{attribute 'qualified_only'}
VAR_GLOBAL
	// Schnittstellenvariablen 
		// System: 
		SystemState								:eSystemState; 
		SystemCommand							:eSystemCommand; 
		Error									:BOOL;
		
		// Kontrollvariablen: 
		Reset									:BOOL;
		
		// Prozessvariablen
		eKraftLimitValue						:sKraftVariablen;
		eKraftErreichtValue						:sKraftVariablen;
		
		
		// SkillStates
		
		// ObjectStates
		Robot_State								:eObjectState;
		Greifer_State							:eObjectState;
		Sensor_State							:eObjectState;
		
			
		
		
		
END_VAR

(* stored: Version 1.1.0.1
   GVL GVL: Id {60ef8ccc-00cf-4757-a644-383c87ef5c44} *)
